ABB RobotStudio station: rsMotion.rspag

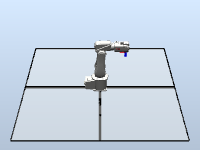
--- station ---
Station rsMotion (saved by RobotStudio 6.7.7936.1011)
Controller rsMotion
  mechanical unit ROB_1: IRB120_3_58__01, 6 joints, base frame (0, 0, 0) mm
Layout (positions relative to the parent item):
  - IRB120_3_58__01 [mechanism, from Robots\IRB120_3_58_G_01.rslib] at (0, 0, 0) mm; joint values [0, 0.0748, -0.0773, 0, 1.5733, 0] (rad or m)
Targets, tools, work objects and paths stored in the station and not in the controller backup, written as RAPID:
! task T_ROB1
MODULE BASE
  PERS tooldata tool1:=[TRUE,[[0,0,0],[1,0,0,0]],[0.001,[0,0,0.001],[1,0,0,0],0,0,0]];
  PERS tooldata tool2:=[TRUE,[[0,0,0],[1,0,0,0]],[0.001,[0,0,0.001],[1,0,0,0],0,0,0]];
  PERS wobjdata wobj1:=[FALSE,TRUE,"",[[0,0,0],[1,0,0,0]],[[0,0,0],[1,0,0,0]]];
  PERS wobjdata wobj2:=[FALSE,TRUE,"",[[0,0,0],[1,0,0,0]],[[0,0,0],[1,0,0,0]]];
ENDMODULE


--- station ---
Station rsMotion (saved by RobotStudio 6.7.7936.1011)
Controller rsMotion
  mechanical unit ROB_1: IRB120_3_58__01, 6 joints, base frame (0, 0, 0) mm
Layout (positions relative to the parent item):
  - IRB120_3_58__01 [mechanism, from Robots\IRB120_3_58_G_01.rslib] at (0, 0, 0) mm; joint values [0, 0.0748, -0.0773, 0, 1.5733, 0] (rad or m)
Targets, tools, work objects and paths stored in the station and not in the controller backup, written as RAPID:
! task T_ROB1
MODULE BASE
  PERS tooldata tool1:=[TRUE,[[0,0,0],[1,0,0,0]],[0.001,[0,0,0.001],[1,0,0,0],0,0,0]];
  PERS tooldata tool2:=[TRUE,[[0,0,0],[1,0,0,0]],[0.001,[0,0,0.001],[1,0,0,0],0,0,0]];
  PERS wobjdata wobj1:=[FALSE,TRUE,"",[[0,0,0],[1,0,0,0]],[[0,0,0],[1,0,0,0]]];
  PERS wobjdata wobj2:=[FALSE,TRUE,"",[[0,0,0],[1,0,0,0]],[[0,0,0],[1,0,0,0]]];
ENDMODULE


--- Backups/rsMotion/RAPID/TASK1/PROGMOD/Module1.mod ---
MODULE Module1
    VAR socketdev server_socket;
    VAR socketdev client_socket;
    VAR string client_ip;

    VAR num nERROR_SUCCESS:=0;
    VAR num nERROR_INVALID_FUNCTION:=1;
    VAR num nERROR_SIGNAL_NOT_FOUND:=2;
    VAR num nERROR_NORUNUNIT:=3;
    VAR num nERROR_NO_ALIASIO_DEF:=4;
    VAR num nERROR_ABORT:=38;
    VAR num nERROR_OUT_OF_RANGE:=84;
    VAR num nERROR_INVALID_PARAMETER:=87;
    VAR num nERROR_TIMEOUT:=88;


    pers wobjdata wWobj;
    pers tooldata tTool;


    PROC main()
        VAR string sParameters{15};
        VAR string sRequest;
        VAR num nCount:=0;
        VAR string sReturn;
        VAR string sResponse;


        SocketCreate server_socket;
        SocketBind server_socket,"172.20.10.14",2001;
        SocketListen server_socket;

        WHILE TRUE DO
            SocketClose client_socket;
            SocketAccept server_socket,client_socket\ClientAddress:=client_ip;
            SocketReceive client_socket\Str:=sRequest;

            IF StrLen(sRequest)>0 THEN
                splitString sRequest,",",sParameters,nCount;
                IF nCount>0 THEN
                    TEST sParameters{1}
                    CASE "robotmovej":
                        RobotMove sParameters,nCount,sReturn;
                    CASE "robotmovel":
                        RobotMove sParameters,nCount,sReturn;
                    CASE "robotmoveabsj":
                        RobotMoveAbsJ sParameters,nCount,sReturn;
                    CASE "robotrotate":
                        RobotRotate sParameters,nCount,sReturn;
                    CASE "robothere":
                        RobotHere sParameters,nCount,sReturn;
                    CASE "robotherej":
                        RobotHerej sParameters,nCount,sReturn;
                    CASE "clamperon":
                        GripperOn sParameters,nCount,sReturn;
                    CASE "clamperoff":
                        GripperOff sParameters,nCount,sReturn;
                    DEFAULT:
                        sReturn:=ValToStr(nERROR_INVALID_PARAMETER);
                    ENDTEST

                    sReturn:=sParameters{1}+","+sReturn;
                    SocketSend client_socket\Str:=sReturn;
                ENDIF
            ENDIF

        ENDWHILE
    ERROR
        RETRY;
    UNDO

    ENDPROC

    PROC splitString(string sString,string s_Seperator,INOUT string sElements{*},inout num nCount)
        VAR num startBit{15};
        VAR num endBit{15};
        VAR num lenBit{15};
        FOR i FROM 1 TO 15 DO
            IF i=1 THEN
                startBit{1}:=1;
            ELSE
                startBit{i}:=endBit{i-1}+1;
                IF startBit{i}>=StrLen(sString) THEN
                    RETURN ;
                ENDIF
            ENDIF

            endBit{i}:=strFind(sString,startBit{i},s_Seperator);
            lenBit{i}:=endBit{i}-startBit{i};
            sElements{i}:=StrPart(sString,startBit{i},lenBit{i});
            nCount:=nCount+1;
        ENDFOR
    ENDPROC

    PROC RobotHere(INOUT string sElements{*},num nCount,inout string sReturn)
        VAR num nFrameIndex;
        VAR num nGripperType;
        VAR robtarget pCurPos;
        VAR bool flag;



        sReturn:=ValToStr(nERROR_INVALID_PARAMETER);
        IF (nCount>=3) THEN
            flag:=StrToVal(sElements{2},nFrameIndex);
            TEST nFrameIndex
            CASE 0:
                wWobj:=wobj0;
            CASE 1:
                wWobj:=wobj1;
            CASE 2:
                wWobj:=wobj2;
            DEFAULT:
                RETURN ;
            ENDTEST

            flag:=StrToVal(sElements{3},nGripperType);

            TEST nGripperType
            CASE 0:
                tTool:=tool0;
            CASE 1:
                tTool:=tool1;
            CASE 2:
                tTool:=tool2;
            DEFAULT:
                RETURN ;
            ENDTEST

            pCurPos:=CRobT(\Tool:=tTool\WObj:=wWobj);
            sReturn:=ValToStr(nERROR_SUCCESS)+",";
            sReturn:=sReturn+ValToStr(Round(pCurPos.trans.x\Dec:=1))+",";
            sReturn:=sReturn+ValToStr(Round(pCurPos.trans.y\Dec:=1))+",";
            sReturn:=sReturn+ValToStr(Round(pCurPos.trans.z\Dec:=1))+",";
            sReturn:=sReturn+ValToStr(Round(pCurPos.rot.q1\Dec:=1))+",";
            sReturn:=sReturn+ValToStr(Round(pCurPos.rot.q2\Dec:=1))+",";
            sReturn:=sReturn+ValToStr(Round(pCurPos.rot.q3\Dec:=1))+",";
            sReturn:=sReturn+ValToStr(Round(pCurPos.rot.q4\Dec:=1))+",";
            sReturn:=sReturn+ValToStr(Round(pCurPos.rot.q4\Dec:=1))+",";
            sReturn:=sReturn+ValToStr(Round(pCurPos.robconf.cf1\Dec:=1))+",";
            sReturn:=sReturn+ValToStr(Round(pCurPos.robconf.cf4\Dec:=1))+",";
            sReturn:=sReturn+ValToStr(Round(pCurPos.robconf.cf6\Dec:=1))+",";
            sReturn:=sReturn+ValToStr(Round(pCurPos.robconf.cfx\Dec:=1))+",";

        ENDIF

    ENDPROC

    PROC RobotHerej(INOUT string sElements{*},num nCount,inout string sReturn)
        VAR jointtarget jCurPos;
        VAR bool flag;

        sReturn:=ValToStr(nERROR_INVALID_PARAMETER);
        IF (nCount>=1) THEN
            jCurPos:=CJointT();
            sReturn:=ValToStr(nERROR_SUCCESS)+",";
            sReturn:=sReturn+ValToStr(jCurPos.robax.rax_1)+",";
            sReturn:=sReturn+ValToStr(jCurPos.robax.rax_2)+",";
            sReturn:=sReturn+ValToStr(jCurPos.robax.rax_3)+",";
            sReturn:=sReturn+ValToStr(jCurPos.robax.rax_4)+",";
            sReturn:=sReturn+ValToStr(jCurPos.robax.rax_5)+",";
            sReturn:=sReturn+ValToStr(jCurPos.robax.rax_6);
        ENDIF

    ENDPROC

    PROC RobotRotate(INOUT string sElements{*},num nCount,inout string sReturn)
        VAR num nRotateDegree;
        VAR jointtarget jCurPos;
        VAR bool flag;
        sReturn:=ValToStr(nERROR_INVALID_PARAMETER);
        IF (nCount>=2) THEN
            flag:=StrToVal(sElements{2},nRotateDegree);
        ENDIF

        jCurPos:=CJointT();
        jCurPos.robax.rax_1:=jCurPos.robax.rax_1+nRotateDegree;
        MoveAbsJ jCurPos,v1000,z50,tool0;

        sReturn:=ValToStr(nERROR_SUCCESS);

    ENDPROC

    PROC RobotMove(INOUT string sElements{*},num nCount,inout string sReturn)
        VAR num nFrameIndex;
        VAR num nGripperType;
        VAR num nPoint{11};
        VAR robtarget pTarget;
        VAR bool flag;
        pTarget.extax:=[9E9,9E9,9E9,9E9,9E9,9E9];


        sReturn:=ValToStr(nERROR_INVALID_PARAMETER);
        IF (nCount>=14) THEN
            FOR i FROM 2 TO 12 DO
                flag:=StrToVal(sElements{i},nPoint{i-1});
            ENDFOR
            pTarget.trans.x:=nPoint{1};
            pTarget.trans.y:=nPoint{2};
            pTarget.trans.z:=nPoint{3};
            pTarget.rot.q1:=nPoint{4};
            pTarget.rot.q2:=nPoint{5};
            pTarget.rot.q3:=nPoint{6};
            pTarget.rot.q4:=nPoint{7};
            pTarget.robconf.cf1:=nPoint{8};
            pTarget.robconf.cf4:=nPoint{9};
            pTarget.robconf.cf6:=nPoint{10};
            pTarget.robconf.cfx:=nPoint{11};


            flag:=StrToVal(sElements{13},nFrameIndex);
            TEST nFrameIndex
            CASE 0:
                wWobj:=wobj0;
            CASE 1:
                wWobj:=wobj1;
            CASE 2:
                wWobj:=wobj2;
            DEFAULT:
                RETURN ;
            ENDTEST

            flag:=StrToVal(sElements{14},nGripperType);
            TEST nGripperType
            CASE 0:
                tTool:=tool0;
            CASE 1:
                tTool:=tool1;
            CASE 2:
                tTool:=tool2;
            DEFAULT:
                RETURN ;
            ENDTEST

            IF sElements{1}="robotmovel" THEN
                MoveL pTarget,v1000,z50,tTool\WObj:=wWobj;
            ELSEIF sElements{1}="robotmovej" THEN
                Movej pTarget,v1000,z50,tTool\WObj:=wWobj;
            ENDIF
        ENDIF

        sReturn:=ValToStr(nERROR_SUCCESS);

    ENDPROC

    PROC RobotMoveAbsJ(INOUT string sElements{*},num nCount,inout string sReturn)
        VAR num nPoint{6};
        VAR jointtarget jTarget;
        VAR bool flag;
        jTarget.extax:=[9E9,9E9,9E9,9E9,9E9,9E9];

        sReturn:=ValToStr(nERROR_INVALID_PARAMETER);
        IF (nCount>=7) THEN
            FOR i FROM 2 TO 7 DO
                flag:=StrToVal(sElements{i},nPoint{i-1});
            ENDFOR
            jTarget.robax.rax_1:=nPoint{1};
            jTarget.robax.rax_2:=nPoint{2};
            jTarget.robax.rax_3:=nPoint{3};
            jTarget.robax.rax_4:=nPoint{4};
            jTarget.robax.rax_5:=nPoint{5};
            jTarget.robax.rax_6:=nPoint{6};

            MoveAbsJ jTarget,v1000,z50,tool0;
        ENDIF

        sReturn:=ValToStr(nERROR_SUCCESS);

    ENDPROC


    PROC GripperOn(INOUT string sElements{*},num nCount,inout string sReturn)
        sReturn:=ValToStr(nERROR_INVALID_PARAMETER);
        IF(nCount>=1) THEN
            set do1;
        ENDIF
        WaitDO do1,1\MaxTime:=20;
        sReturn:=ValToStr(nERROR_SUCCESS);
        ERROR
        IF ERRNO=ERR_WAIT_MAXTIME THEN
            sReturn:=ValToStr(nERROR_TIMEOUT);
        ELSEIF ERRNO=ERR_SIG_NOT_VALID THEN
            sReturn:=ValToStr(nERROR_SIGNAL_NOT_FOUND);
        ELSEIF ERRNO=ERR_NORUNUNIT THEN
            sReturn:=ValToStr(nERROR_NORUNUNIT);
        ELSEIF ERRNO=ERR_NO_ALIASIO_DEF THEN
            sReturn:=ValToStr(nERROR_NO_ALIASIO_DEF);
        ENDIF


    ENDPROC


    PROC GripperOff(INOUT string sElements{*},num nCount,inout string sReturn)
        sReturn:=ValToStr(nERROR_INVALID_PARAMETER);
        IF(nCount>=1) THEN
            Reset do1;
        ENDIF
        WaitDO do1,0\MaxTime:=20;
        sReturn:=ValToStr(nERROR_SUCCESS);
        ERROR
        IF ERRNO=ERR_WAIT_MAXTIME THEN
            sReturn:=ValToStr(nERROR_TIMEOUT);
        ELSEIF ERRNO=ERR_SIG_NOT_VALID THEN
            sReturn:=ValToStr(nERROR_SIGNAL_NOT_FOUND);
        ELSEIF ERRNO=ERR_NORUNUNIT THEN
            sReturn:=ValToStr(nERROR_NORUNUNIT);
        ELSEIF ERRNO=ERR_NO_ALIASIO_DEF THEN
            sReturn:=ValToStr(nERROR_NO_ALIASIO_DEF);
        ENDIF


    ENDPROC

ENDMODULE

--- Backups/rsMotion/SYSPAR/EIO.cfg ---
EIO:CFG_1.0:6:1::
#
INDUSTRIAL_NETWORK:

      -Name "DeviceNet" -Label "DeviceNet Master/Slave Network" -Address "2"
#
DEVICENET_DEVICE:

      -Name "Device1" -Simulated
#
DEVICENET_INTERNAL_DEVICE:

      -Name "DN_Internal_Device" -VendorName "ABB Robotics"\
      -ProductName "DeviceNet Internal Slave Device"
#
EIO_SIGNAL:

      -Name "do1" -SignalType "DO" -Device "Device1" -DeviceMap "0"
